PROGRAM MAIN
VAR
END_VAR

END_PROGRAM

(* stored: Version 1.1.0.1, ProductVersion 3.1.0.26
   POU MAIN: Id {dddb9f00-536c-4c41-8309-0f4613f140b5} *)
